(* CODESYS project ParkingRampa.project
   Title: semiraski_awad_i_d
   Version: 0.0.0.0
   Author: CA Simple

Project tree, tasks and I/O mapping:
  MyController : TM238LDD24DT, Schneider Electric, order no. TM238LDD24DT, version 4.0.1.28
      settings: OpcUa Enable = False; Expansion Tasks.Expansion 1 Task Name = 'MAST'
    application Application
      task MAST (cyclic, interval 20 ms, priority 15, watchdog 100 ms x 1) calls POU, rampa_dole, rampa_gore, termickiRelej
      global variables GVL
      program POU [SFC]: Init_entry, Init_active, podizanje_rampe_active, Init_exit, spustanje_rampe_active, podizanje_rampe_exit, spustanje_rampe_exit, motor_crko_active, auta_ima_active, auta_nema_active, cekanje_5_sekundi_active, auta_ima_exit, motor_crko_exit
      program rampa_dole [ST]
      program rampa_gore [ST]
      Symbols
      program termickiRelej [ST]
    Embedded Functions
      IO : IO, Schneider Electric, version 4.0.1.28
          input  iwIO_IW0 : WORD  // IW0
          output qwIO_QW0 : WORD  // QW0
      HSC : HSC, Schneider Electric, version 4.0.1.28
      PTO_PWM : PTO_PWM, Schneider Electric, version 4.0.1.28
    Serial Line
      SoMachine_Network_Manager : SoMachine-Network Manager, Schneider Electric, version 4.0.0.2
    Module_1 : TM2AMI8HT, Schneider Electric, order no. TM2AMI8HT, version 4.0.1.28
        input  Application.potenciometar : INT  // IW0
        input  iiModule_1_IW1 : INT  // IW1
        input  iiModule_1_IW2 : INT  // IW2
        input  iiModule_1_IW3 : INT  // IW3
        input  iiModule_1_IW4 : INT  // IW4
        input  iiModule_1_IW5 : INT  // IW5
        input  iiModule_1_IW6 : INT  // IW6
        input  iiModule_1_IW7 : INT  // IW7
  HMIS5T : HMIS5T, Schneider Electric, order no. HMIS5T, version 3.5.3.54
    HMI Application
    COM1
      SoMachine_Network_Manager1 : SoMachine-Network Manager, Schneider Electric, version 4.0.0.2
    Ethernet
      SoMachine_Network_Manager2 : SoMachine-Network Manager, Schneider Electric, version 4.0.0.2
    USB
      SoMachine_Network_Manager3 : SoMachine-Network Manager, Schneider Electric, version 4.0.0.2
  Vijeo Designer Project Container Data
  Vijeo Designer Project Container
*)

// MyController/Application/GVL
VAR_GLOBAL
	timer_30s_triger: F_TRIG;
	timer_30s: TP;
	okidac_timer_30: BOOL;
	potvrda: BOOL;
	motor: BOOL;
	motor_neg: BOOL;
	motor_poz: BOOL;
	potenciometar: INT;
	senzor: BOOL;
	taster: BOOL;
	polozaj_dole: BOOL;
	polozaj_gore: BOOL;
	timer_triger: F_TRIG;
	timer_5s: TP;
	vrijeme_dana: TIME;
	ima_auto: BOOL;
	okidac_senzor: BOOL;
	pom: BOOL := FALSE;
	ima_papir: BOOL := TRUE;
	radi_motor: BOOL := TRUE;
	potvrda_preuzeta: BOOL;
	Termicki_relej: BOOL;
	start: BOOL;
	hitan_stop: BOOL;
	pocetak: BOOL;
END_VAR

// MyController/Application/POU
PROGRAM POU

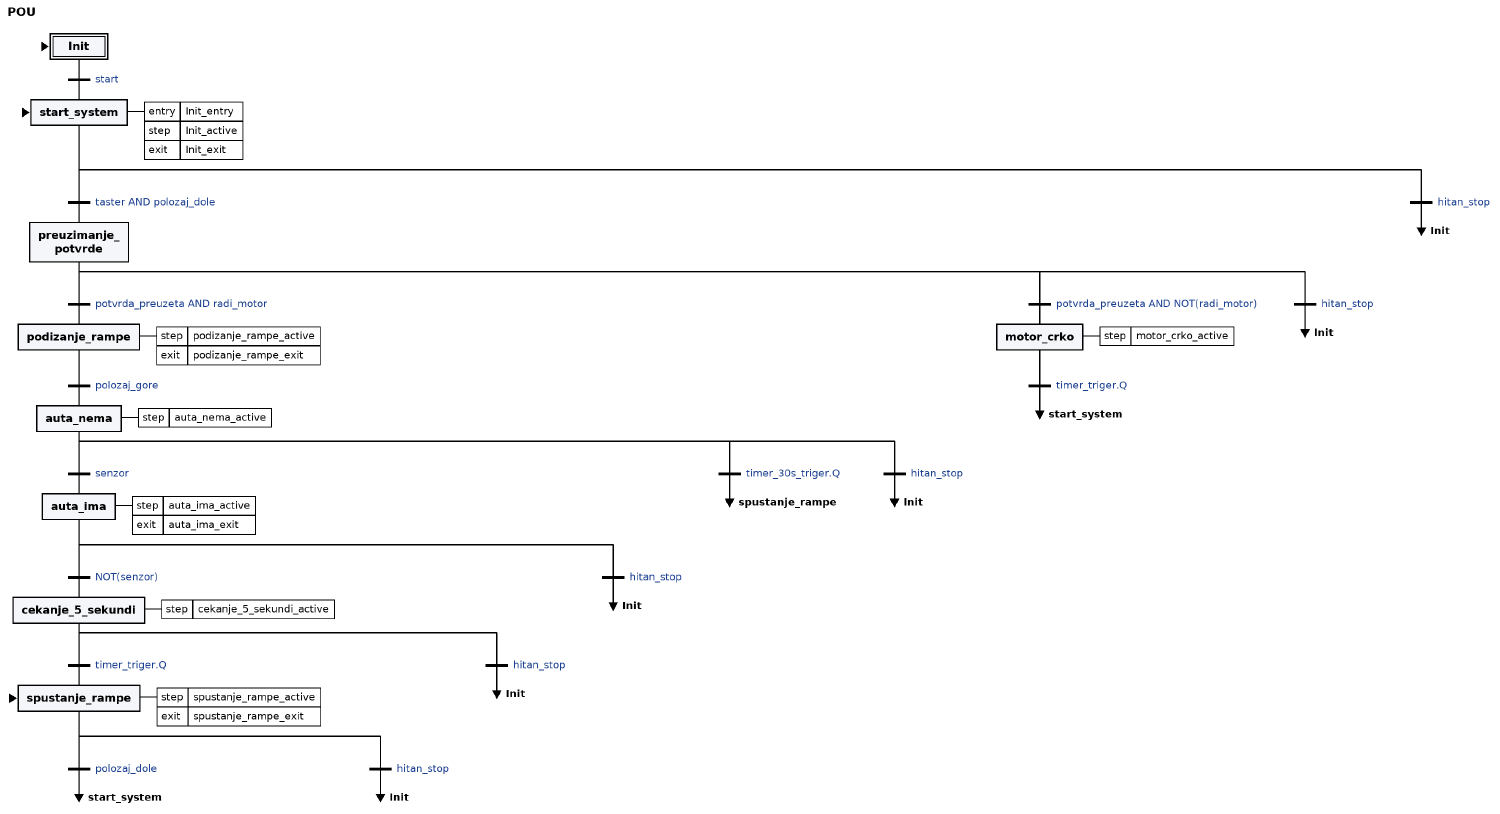
INITIAL_STEP Init:
END_STEP
TRANSITION FROM Init TO start_system
    := start;
END_TRANSITION
STEP start_system:
    Init_entry(P1);  // entry action
    Init_active(N);  // step action
    Init_exit(P0);  // exit action
END_STEP
TRANSITION FROM start_system TO preuzimanje_potvrde
    := taster AND polozaj_dole;
END_TRANSITION
TRANSITION FROM start_system TO Init
    := hitan_stop;
END_TRANSITION
STEP preuzimanje_potvrde:
END_STEP
TRANSITION FROM preuzimanje_potvrde TO podizanje_rampe
    := potvrda_preuzeta AND radi_motor;
END_TRANSITION
STEP podizanje_rampe:
    podizanje_rampe_active(N);  // step action
    podizanje_rampe_exit(P0);  // exit action
END_STEP
TRANSITION FROM podizanje_rampe TO auta_nema
    := polozaj_gore;
END_TRANSITION
TRANSITION FROM preuzimanje_potvrde TO motor_crko
    := potvrda_preuzeta AND NOT(radi_motor);
END_TRANSITION
STEP motor_crko:
    motor_crko_active(N);  // step action
END_STEP
TRANSITION FROM motor_crko TO start_system
    := timer_triger.Q;
END_TRANSITION
TRANSITION FROM preuzimanje_potvrde TO Init
    := hitan_stop;
END_TRANSITION
STEP auta_nema:
    auta_nema_active(N);  // step action
END_STEP
TRANSITION FROM auta_nema TO auta_ima
    := senzor;
END_TRANSITION
TRANSITION FROM auta_nema TO spustanje_rampe
    := timer_30s_triger.Q;
END_TRANSITION
TRANSITION FROM auta_nema TO Init
    := hitan_stop;
END_TRANSITION
STEP auta_ima:
    auta_ima_active(N);  // step action
    auta_ima_exit(P0);  // exit action
END_STEP
TRANSITION FROM auta_ima TO cekanje_5_sekundi
    := NOT(senzor);
END_TRANSITION
TRANSITION FROM auta_ima TO Init
    := hitan_stop;
END_TRANSITION
STEP cekanje_5_sekundi:
    cekanje_5_sekundi_active(N);  // step action
END_STEP
TRANSITION FROM cekanje_5_sekundi TO spustanje_rampe
    := timer_triger.Q;
END_TRANSITION
TRANSITION FROM cekanje_5_sekundi TO Init
    := hitan_stop;
END_TRANSITION
STEP spustanje_rampe:
    spustanje_rampe_active(N);  // step action
    spustanje_rampe_exit(P0);  // exit action
END_STEP
TRANSITION FROM spustanje_rampe TO start_system
    := polozaj_dole;
END_TRANSITION
TRANSITION FROM spustanje_rampe TO Init
    := hitan_stop;
END_TRANSITION

ACTION Init_entry:
motor_poz := FALSE;
motor_neg := FALSE;
motor := FALSE;
potvrda := FALSE;
potvrda_preuzeta := FALSE;
start := FALSE;
hitan_stop := FALSE;

okidac_senzor := FALSE;
okidac_timer_30 := FALSE;
timer_triger ( CLK := pom );
timer_30s_triger ( CLK := pom );

timer_5s (IN := pom);

pocetak := TRUE;
END_ACTION

ACTION Init_active:
IF potenciometar > 257 THEN
	motor_neg := TRUE;
	WHILE potenciometar > 255 DO
		potenciometar := potenciometar - 1;
	END_WHILE;
END_IF;
motor_neg := FALSE;

IF potenciometar < 254 THEN
	motor_poz := TRUE;
	WHILE potenciometar < 255 DO	
		potenciometar := potenciometar + 1;
	END_WHILE;
END_IF;
motor_poz := FALSE;
END_ACTION

ACTION podizanje_rampe_active:
motor := TRUE;
motor_poz := TRUE;	
WHILE potenciometar <= 511 DO
	potenciometar := potenciometar + 1;
END_WHILE;
END_ACTION

ACTION Init_exit:
motor := FALSE;
motor_poz := FALSE;
motor_neg := FALSE;

potvrda := TRUE;
vrijeme_dana := TIME();

pocetak := FALSE;
END_ACTION

ACTION spustanje_rampe_active:
motor := TRUE;
motor_neg := TRUE;	
WHILE potenciometar >= 255 DO
	potenciometar := potenciometar - 1;
END_WHILE;
END_ACTION

ACTION podizanje_rampe_exit:
motor_poz := FALSE;
motor := FALSE;
okidac_timer_30 := TRUE;
END_ACTION

ACTION spustanje_rampe_exit:
motor_neg := FALSE;
motor := FALSE;
END_ACTION

ACTION motor_crko_active:
okidac_senzor := TRUE;
timer_5s (IN := okidac_senzor, PT := T#5S);

timer_triger ( CLK := timer_5s.Q );
okidac_senzor := FALSE;
END_ACTION

ACTION auta_ima_active:

END_ACTION

ACTION auta_nema_active:
timer_30s (IN := okidac_timer_30, PT := T#30S);

timer_30s_triger ( CLK := timer_30s.Q );
okidac_timer_30 := FALSE;
END_ACTION

ACTION cekanje_5_sekundi_active:
timer_5s (IN := okidac_senzor, PT := T#5S);

timer_triger ( CLK := timer_5s.Q );
okidac_senzor := FALSE;
END_ACTION

ACTION auta_ima_exit:
okidac_senzor := TRUE;
END_ACTION

ACTION motor_crko_exit:

END_ACTION

END_PROGRAM

// MyController/Application/rampa_dole
PROGRAM rampa_dole
VAR
END_VAR

IF (potenciometar >= 254 AND potenciometar <= 257) THEN
	polozaj_dole := TRUE;
ELSE 
	polozaj_dole := FALSE;
END_IF;

END_PROGRAM

// MyController/Application/rampa_gore
PROGRAM rampa_gore
VAR
END_VAR

IF (potenciometar >= 510 AND potenciometar <= 512) THEN
	polozaj_gore := TRUE;
ELSE 
	polozaj_gore := FALSE;
END_IF;

END_PROGRAM

// MyController/Application/termickiRelej
PROGRAM termickiRelej
VAR
END_VAR

IF Termicki_relej=TRUE THEN
	radi_motor := FALSE;
END_IF

END_PROGRAM
